TYPE ST_IvekCyclicInput :
STRUCT
	// Controller -> PLC. Link these members to EDS-generated input tags.
    udiStatusFlags       : UDINT;
    udiStatusFlagsExt    : UDINT;
    eStatusState         : E_IvekStatusState;
    udiFaultCode         : UDINT;
    udiAlertCode         : UDINT;
    usiCurrentRecipe     : USINT;
END_STRUCT
END_TYPE

(* stored: Version 1.1.0.1, ProductVersion 3.1.4026.18
   DUT ST_IvekCyclicInput: Id {602d1742-6dd6-43e3-a59a-0b71eeaef8a2} *)
